// Unfinished, and excluded from the build (the POUs\Drafts folder has
// ExcludeFromBuild): the project compiles without it.
FUNCTION_BLOCK FB_Draft
VAR
    nValue : DINT;
END_VAR

nValue :=

END_FUNCTION_BLOCK

(* stored: Version 1.1.0.1, ProductVersion 3.1.4024.12
   POU FB_Draft: Id {5f1c2d9e-0a6b-4c11-9d3e-7a1b2c3d4e70}, SpecialFunc None *)
